ABB RAPID module: Module1.mod

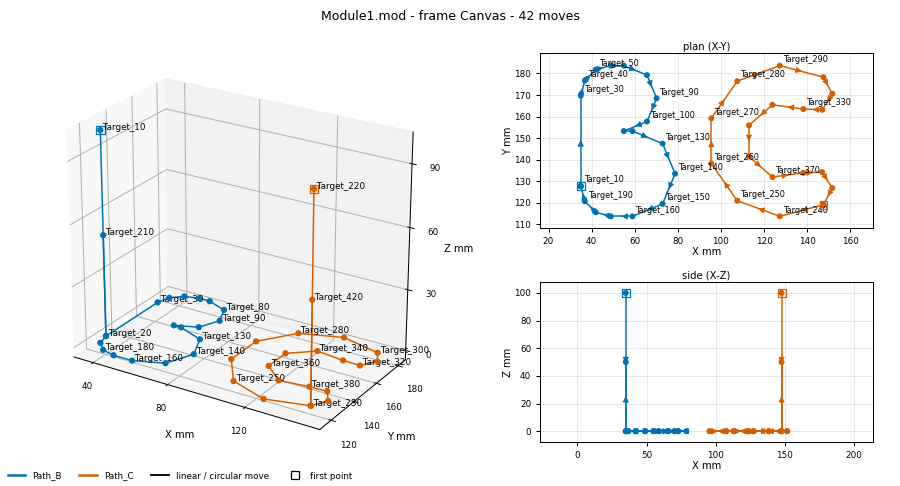
[picture p0: tool path of Module1.mod in frame Canvas, 42 of 44 moves have a stored position in this frame; points joined in program order, loops and branches not executed]
MODULE Module1
    CONST robtarget Target_10:=[[34.951366553,127.686109727,100.000011021],[0.000000111,-0.505561819,0.862790384,0.000000254],[0,0,0,0],[9E+09,9E+09,9E+09,9E+09,9E+09,9E+09]];
    CONST robtarget Target_20:=[[34.951421709,127.68610326,0.000011021],[0.000000111,-0.505561819,0.862790384,0.000000254],[0,0,0,0],[9E+09,9E+09,9E+09,9E+09,9E+09,9E+09]];
    CONST robtarget Target_30:=[[34.951446662,169.68610326,0.000008305],[0.000000111,-0.505561819,0.862790384,0.000000254],[0,0,0,0],[9E+09,9E+09,9E+09,9E+09,9E+09,9E+09]];
    CONST robtarget Target_40:=[[36.827095167,176.686102147,0.000008887],[0.000000223,-0.505561758,0.86279042,0.000000165],[0,0,0,0],[9E+09,9E+09,9E+09,9E+09,9E+09,9E+09]];
    CONST robtarget Target_50:=[[41.951453865,181.810454755,0.000011381],[0.000000276,-0.505561694,0.862790457,0.000000031],[0,0,0,0],[9E+09,9E+09,9E+09,9E+09,9E+09,9E+09]];
    CONST robtarget Target_60:=[[48.951454979,183.686094943,0.000015122],[0.000000254,-0.505561644,0.862790487,-0.000000112],[0,0,0,0],[9E+09,9E+09,9E+09,9E+09,9E+09,9E+09]];
    CONST robtarget Target_70:=[[54.951454979,183.686091378,0.000018431],[0.000000254,-0.505561644,0.862790487,-0.000000112],[0,0,0,0],[9E+09,9E+09,9E+09,9E+09,9E+09,9E+09]];
    CONST robtarget Target_80:=[[65.711772914,179.229014265,0.000024654],[0.000000101,-0.505561621,0.8627905,-0.000000258],[0,0,0,0],[9E+09,9E+09,9E+09,9E+09,9E+09,9E+09]];
    CONST robtarget Target_90:=[[70.168837242,168.468691033,0.000027808],[0.000000221,-0.505561629,0.862790495,-0.000000167],[0,0,0,0],[9E+09,9E+09,9E+09,9E+09,9E+09,9E+09]];
    CONST robtarget Target_100:=[[65.711760128,157.708373097,0.000026046],[0.000000222,-0.505561629,0.862790495,-0.000000167],[0,0,0,0],[9E+09,9E+09,9E+09,9E+09,9E+09,9E+09]];
    CONST robtarget Target_110:=[[54.951436897,153.25130877,0.000020398],[0.000000222,-0.505561629,0.862790495,-0.000000167],[0,0,0,0],[9E+09,9E+09,9E+09,9E+09,9E+09,9E+09]];
    CONST robtarget Target_120:=[[58.951436897,153.251306393,0.000022605],[0.000000222,-0.505561629,0.862790495,-0.000000167],[0,0,0,0],[9E+09,9E+09,9E+09,9E+09,9E+09,9E+09]];
    CONST robtarget Target_130:=[[72.939850213,147.457106145,0.000030695],[0.000000101,-0.505561621,0.8627905,-0.000000258],[0,0,0,0],[9E+09,9E+09,9E+09,9E+09,9E+09,9E+09]];
    CONST robtarget Target_140:=[[78.734033839,133.468685944,0.000034796],[0.000000221,-0.505561629,0.862790495,-0.000000167],[0,0,0,0],[9E+09,9E+09,9E+09,9E+09,9E+09,9E+09]];
    CONST robtarget Target_150:=[[72.939833591,119.480272628,0.000032505],[0.000000222,-0.505561629,0.862790495,-0.000000167],[0,0,0,0],[9E+09,9E+09,9E+09,9E+09,9E+09,9E+09]];
    CONST robtarget Target_160:=[[58.951413391,113.686089002,0.000025164],[0.000000222,-0.505561629,0.862790495,-0.000000167],[0,0,0,0],[9E+09,9E+09,9E+09,9E+09,9E+09,9E+09]];
    CONST robtarget Target_170:=[[48.95141339,113.686094943,0.000019648],[0.000000222,-0.505561629,0.862790495,-0.000000167],[0,0,0,0],[9E+09,9E+09,9E+09,9E+09,9E+09,9E+09]];
    CONST robtarget Target_180:=[[41.951414505,115.561743448,0.000015666],[0.000000222,-0.505561629,0.862790495,-0.000000168],[0,0,0,0],[9E+09,9E+09,9E+09,9E+09,9E+09,9E+09]];
    CONST robtarget Target_190:=[[36.827061896,120.686102146,0.000012509],[0.000000222,-0.505561629,0.862790495,-0.000000167],[0,0,0,0],[9E+09,9E+09,9E+09,9E+09,9E+09,9E+09]];
    CONST robtarget Target_200:=[[34.951421709,127.68610326,0.000011021],[0.000000111,-0.505561819,0.862790384,0.000000254],[0,0,0,0],[9E+09,9E+09,9E+09,9E+09,9E+09,9E+09]];
    CONST robtarget Target_210:=[[34.95139413,127.686106494,50.000011021],[0.000000111,-0.505561819,0.862790384,0.000000254],[0,0,0,0],[9E+09,9E+09,9E+09,9E+09,9E+09,9E+09]];
    CONST robtarget Target_220:=[[147.618028106,119.079361862,100.00007372],[0.000000222,-0.505561629,0.862790495,-0.000000168],[0,0,0,0],[9E+09,9E+09,9E+09,9E+09,9E+09,9E+09]];
    CONST robtarget Target_230:=[[147.618083262,119.079355396,0.00007372],[0.000000222,-0.505561629,0.862790495,-0.000000168],[0,0,0,0],[9E+09,9E+09,9E+09,9E+09,9E+09,9E+09]];
    CONST robtarget Target_240:=[[127.307461338,113.724677971,0.000062863],[0.000000222,-0.505561629,0.862790496,-0.000000168],[0,0,0,0],[9E+09,9E+09,9E+09,9E+09,9E+09,9E+09]];
    CONST robtarget Target_250:=[[107.588929901,120.96162838,0.000051519],[0.000000222,-0.505561629,0.862790496,-0.000000168],[0,0,0,0],[9E+09,9E+09,9E+09,9E+09,9E+09,9E+09]];
    CONST robtarget Target_260:=[[95.564281966,138.183758774,0.000043774],[0.000000221,-0.50556163,0.862790495,-0.000000167],[0,0,0,0],[9E+09,9E+09,9E+09,9E+09,9E+09,9E+09]];
    CONST robtarget Target_270:=[[95.564294445,159.188375725,0.000042415],[0.000000182,-0.505561785,0.862790404,0.000000209],[0,0,0,0],[9E+09,9E+09,9E+09,9E+09,9E+09,9E+09]];
    CONST robtarget Target_280:=[[107.588962844,176.41049183,0.000047934],[0.000000269,-0.50556171,0.862790448,0.000000067],[0,0,0,0],[9E+09,9E+09,9E+09,9E+09,9E+09,9E+09]];
    CONST robtarget Target_290:=[[127.30750288,183.647418809,0.000058341],[0.000000259,-0.505561647,0.862790485,-0.000000099],[0,0,0,0],[9E+09,9E+09,9E+09,9E+09,9E+09,9E+09]];
    CONST robtarget Target_300:=[[147.618118442,178.29271725,0.000069891],[0.000000155,-0.50556162,0.862790501,-0.00000023],[0,0,0,0],[9E+09,9E+09,9E+09,9E+09,9E+09,9E+09]];
    CONST robtarget Target_310:=[[151.69481496,170.550427829,0.00007264],[0.000000222,-0.505561629,0.862790496,-0.000000168],[0,0,0,0],[9E+09,9E+09,9E+09,9E+09,9E+09,9E+09]];
    CONST robtarget Target_320:=[[147.028143896,163.148760369,0.000070545],[0.000000221,-0.50556163,0.862790495,-0.000000167],[0,0,0,0],[9E+09,9E+09,9E+09,9E+09,9E+09,9E+09]];
    CONST robtarget Target_330:=[[138.284776313,163.489382332,0.000065699],[0.000000222,-0.505561629,0.862790495,-0.000000167],[0,0,0,0],[9E+09,9E+09,9E+09,9E+09,9E+09,9E+09]];
    CONST robtarget Target_340:=[[123.933920312,165.451325655,0.000057658],[0.000000221,-0.505561629,0.862790495,-0.000000167],[0,0,0,0],[9E+09,9E+09,9E+09,9E+09,9E+09,9E+09]];
    CONST robtarget Target_350:=[[113.020307718,155.92823006,0.000052254],[0.000000221,-0.50556163,0.862790495,-0.000000167],[0,0,0,0],[9E+09,9E+09,9E+09,9E+09,9E+09,9E+09]];
    CONST robtarget Target_360:=[[113.020299112,141.443883696,0.000053191],[0.000000004,-0.505561636,0.862790492,-0.000000278],[0,0,0,0],[9E+09,9E+09,9E+09,9E+09,9E+09,9E+09]];
    CONST robtarget Target_370:=[[123.933900391,131.920775133,0.000059826],[0.000000212,-0.505561627,0.862790497,-0.00000018],[0,0,0,0],[9E+09,9E+09,9E+09,9E+09,9E+09,9E+09]];
    CONST robtarget Target_380:=[[138.284758724,133.882701404,0.000067614],[0.000000275,-0.505561699,0.862790455,0.000000042],[0,0,0,0],[9E+09,9E+09,9E+09,9E+09,9E+09,9E+09]];
    CONST robtarget Target_390:=[[147.02812671,134.223312978,0.000072415],[0.000000173,-0.505561621,0.8627905,-0.000000217],[0,0,0,0],[9E+09,9E+09,9E+09,9E+09,9E+09,9E+09]];
    CONST robtarget Target_400:=[[151.694788979,126.821639973,0.000075468],[-0.000000102,-0.505561668,0.862790473,-0.000000258],[0,0,0,0],[9E+09,9E+09,9E+09,9E+09,9E+09,9E+09]];
    CONST robtarget Target_410:=[[147.618083262,119.079355396,0.00007372],[0.000000222,-0.505561629,0.862790495,-0.000000168],[0,0,0,0],[9E+09,9E+09,9E+09,9E+09,9E+09,9E+09]];
    CONST robtarget Target_420:=[[147.618055684,119.079358628,50.00007372],[0.000000222,-0.505561629,0.862790495,-0.000000168],[0,0,0,0],[9E+09,9E+09,9E+09,9E+09,9E+09,9E+09]];
    CONST jointtarget Start:=[[0,0,0,0,30,0],[9E+09,9E+09,9E+09,9E+09,9E+09,9E+09]];
    CONST jointtarget Middle:=[[0,30,0,50,50,0],[9E+09,9E+09,9E+09,9E+09,9E+09,9E+09]];
    PROC main()
        Path_Start;
        Path_Middle;
        Path_B;
        Path_C;
        Path_Middle;
        Path_Start;
    ENDPROC
    PROC Path_B()
        MoveL Target_10,v60,z50,MarkerTool\WObj:=Canvas;
        MoveL Target_20,v60,z50,MarkerTool\WObj:=Canvas;
        MoveL Target_30,v60,z50,MarkerTool\WObj:=Canvas;
        MoveL Target_40,v60,z50,MarkerTool\WObj:=Canvas;
        MoveL Target_50,v60,z50,MarkerTool\WObj:=Canvas;
        MoveL Target_60,v60,z50,MarkerTool\WObj:=Canvas;
        MoveL Target_70,v60,z50,MarkerTool\WObj:=Canvas;
        MoveL Target_80,v60,z50,MarkerTool\WObj:=Canvas;
        MoveL Target_90,v60,z50,MarkerTool\WObj:=Canvas;
        MoveL Target_100,v60,z50,MarkerTool\WObj:=Canvas;
        MoveL Target_110,v60,z50,MarkerTool\WObj:=Canvas;
        MoveL Target_120,v60,z50,MarkerTool\WObj:=Canvas;
        MoveL Target_130,v60,z50,MarkerTool\WObj:=Canvas;
        MoveL Target_140,v60,z50,MarkerTool\WObj:=Canvas;
        MoveL Target_150,v60,z50,MarkerTool\WObj:=Canvas;
        MoveL Target_160,v60,z50,MarkerTool\WObj:=Canvas;
        MoveL Target_170,v60,z50,MarkerTool\WObj:=Canvas;
        MoveL Target_180,v60,z50,MarkerTool\WObj:=Canvas;
        MoveL Target_190,v60,z50,MarkerTool\WObj:=Canvas;
        MoveL Target_200,v60,z50,MarkerTool\WObj:=Canvas;
        MoveL Target_210,v60,z50,MarkerTool\WObj:=Canvas;
    ENDPROC
    PROC Path_C()
        MoveL Target_220,v100,z50,MarkerTool\WObj:=Canvas;
        MoveL Target_230,v100,z50,MarkerTool\WObj:=Canvas;
        MoveL Target_240,v100,z50,MarkerTool\WObj:=Canvas;
        MoveL Target_250,v100,z50,MarkerTool\WObj:=Canvas;
        MoveL Target_260,v100,z50,MarkerTool\WObj:=Canvas;
        MoveL Target_270,v100,z50,MarkerTool\WObj:=Canvas;
        MoveL Target_280,v100,z50,MarkerTool\WObj:=Canvas;
        MoveL Target_290,v100,z50,MarkerTool\WObj:=Canvas;
        MoveL Target_300,v100,z50,MarkerTool\WObj:=Canvas;
        MoveL Target_310,v100,z50,MarkerTool\WObj:=Canvas;
        MoveL Target_320,v100,z50,MarkerTool\WObj:=Canvas;
        MoveL Target_330,v100,z50,MarkerTool\WObj:=Canvas;
        MoveL Target_340,v100,z50,MarkerTool\WObj:=Canvas;
        MoveL Target_350,v100,z50,MarkerTool\WObj:=Canvas;
        MoveL Target_360,v100,z50,MarkerTool\WObj:=Canvas;
        MoveL Target_370,v100,z50,MarkerTool\WObj:=Canvas;
        MoveL Target_380,v100,z50,MarkerTool\WObj:=Canvas;
        MoveL Target_390,v100,z50,MarkerTool\WObj:=Canvas;
        MoveL Target_400,v100,z50,MarkerTool\WObj:=Canvas;
        MoveL Target_410,v100,z50,MarkerTool\WObj:=Canvas;
        MoveL Target_420,v100,z50,MarkerTool\WObj:=Canvas;
    ENDPROC
    PROC Path_Start()
        MoveAbsJ Start,v300,z100,MarkerTool\WObj:=Canvas;
    ENDPROC
    PROC Path_Middle()
        MoveAbsJ Middle,v300,z100,MarkerTool\WObj:=Canvas;
    ENDPROC
ENDMODULE
